(* PLC project cmd_single_acting_valve, Dassault Systèmes ControlBuild 2024x *)
(* stored: creationDateTime 2023-10-03T11:13:36-01:00 *)

FUNCTION_BLOCK actuator
  VAR_INPUT
    autoMode : BOOL := false;
    manualMode : BOOL := false;
  END_VAR
  VAR_INPUT
    autoOpenCmd : BOOL := false;
  END_VAR
  VAR_INPUT
    openValvePB : BOOL := false;
  END_VAR
  VAR_INPUT
    generalFault : BOOL := false;
  END_VAR
  VAR_OUTPUT
    openCmd : BOOL := false;
  END_VAR

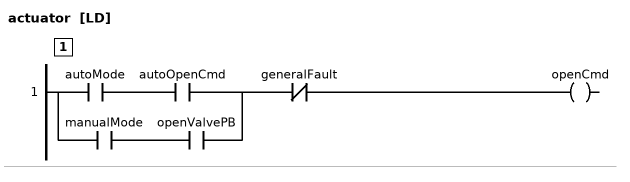
(* LD diagram, written out as Structured Text *)
1:
openCmd := (autoMode AND autoOpenCmd OR manualMode AND openValvePB) AND NOT generalFault;
END_FUNCTION_BLOCK

FUNCTION_BLOCK faults
  VAR_INPUT
    openCmd : BOOL := false;
  END_VAR
  VAR_INPUT
    openedSensorFB : BOOL := false;
    closedSensorFB : BOOL := false;
  END_VAR
  VAR_INPUT
    acknowledgePB : BOOL := false;
  END_VAR
  VAR_OUTPUT
    generalFault : BOOL := false;
  END_VAR
  VAR
    discordanceFault : BOOL := false;
    openedSensorFault : BOOL := false;
    closedSensorFault : BOOL := false;
  END_VAR
  VAR CONSTANT
    presetMvt : TIME := T#0h0m4s0ms;
    presetDiscordance : TIME := T#0h0m0s200ms;
  END_VAR

(* LD diagram, written out as Structured Text *)
1:
IF acknowledgePB THEN discordanceFault := FALSE; END_IF;
IF acknowledgePB THEN openedSensorFault := FALSE; END_IF;
IF acknowledgePB THEN closedSensorFault := FALSE; END_IF;
IF acknowledgePB THEN generalFault := FALSE; END_IF;
2:
TON_O(IN := openCmd, PT := presetMvt);
IF TON_O.Q0 AND NOT openedSensorFB THEN openedSensorFault := TRUE; END_IF;
TON_C(IN := NOT openCmd, PT := presetMvt);
IF TON_C.Q0 AND NOT closedSensorFB THEN closedSensorFault := TRUE; END_IF;
3:
TON_DISC(IN := openedSensorFB AND closedSensorFB, PT := presetDiscordance);
IF TON_DISC.Q0 THEN discordanceFault := TRUE; END_IF;
4:
IF discordanceFault OR openedSensorFault OR closedSensorFault THEN generalFault := TRUE; END_IF;
END_FUNCTION_BLOCK

(* Command of a single acting valve with fault detection *)
PROGRAM cmd_equipment_library.cmd_single_acting_valve
  VAR_INPUT
    autoMode : BOOL := false;
    manualMode : BOOL := false;
  END_VAR
  VAR_INPUT
    autoOpenCmd : BOOL := false;
  END_VAR
  VAR_INPUT
    openValvePB : BOOL := false;
  END_VAR
  VAR_INPUT
    openedSensorFB : BOOL := false;
    closedSensorFB : BOOL := false;
  END_VAR
  VAR_INPUT
    acknowledgePB : BOOL := false;
  END_VAR
  VAR_OUTPUT
    openCmd : BOOL := false;
  END_VAR
  VAR_OUTPUT
    generalFault : BOOL := false;
  END_VAR

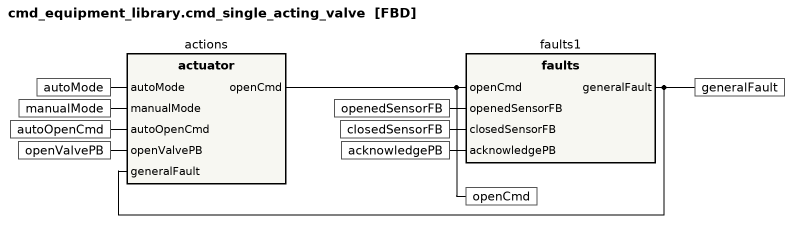
(* FBD diagram, written out as Structured Text *)
faults1(openCmd := actions.openCmd, openedSensorFB := openedSensorFB, closedSensorFB := closedSensorFB, acknowledgePB := acknowledgePB);
actions(autoMode := autoMode, manualMode := manualMode, autoOpenCmd := autoOpenCmd, openValvePB := openValvePB, generalFault := faults1.generalFault);
openCmd := actions.openCmd;
generalFault := faults1.generalFault;
END_PROGRAM
